// TIA Portal V20 export
DATA_BLOCK "ProdDataSimulation"   // DB5
{ DB_Accessible_From_OPC_UA := 'FALSE' }
// stored: DBAccessibleFromOPCUA false, DBAccessibleFromWebserver false, MemoryReserve 100
   VAR
      ProdDataCounter { ExternalAccessible := 'False'; ExternalVisible := 'False'; ExternalWritable := 'False'} : Struct   // Test tag prod data
         ProdDataCounter1Up1 : Bool;   // Test tag prod data
         ProdDataCounter1Up2 : Bool;   // Test tag prod data
         ProdDataCounter1Down1 : Bool;   // Test tag prod data
         ProdDataCounter1Down2 : Bool;   // Test tag prod data
         ProdDataCounter1Reset1 : Bool;   // Test tag prod data
         ProdDataCounter1Reset2 : Bool;   // Test tag prod data
         ProdDataCounter1ResetAll : Bool;   // Test tag prod data
         ProdDataCounter2Up1 : Bool;
         ProdDataCounter2Up2 : Bool;
         ProdDataCounter2Down1 : Bool;
         ProdDataCounter2Down2 : Bool;
         ProdDataCounter2Reset1 : Bool;
         ProdDataCounter2Reset2 : Bool;
         ProdDataCounter2ResetAll : Bool;
         userInterfaceVisibilityDataSet2Counter : DWord := 2#0000_0000_0000_0000_0000_0000_0000_0011;
         userInterfaceVisibilityDataSet1Counter : DWord := 2#0000_0000_0000_0000_0011_1111_1111_1111;
         ProdDataEnable : Bool;
      END_STRUCT;
      ProdDataCyclic { ExternalAccessible := 'False'; ExternalVisible := 'False'; ExternalWritable := 'False'} : Struct   // Test tag prod data
         cycleTimer1Run1 : Bool;   // Test tag prod data
         cycleTimer1Run2 : Bool;   // Test tag prod data
         cycleTimer1Hold1 : Bool;   // Test tag prod data
         cycleTimer1Hold2 : Bool;   // Test tag prod data
         cycleTimer1Reset1 : Bool;   // Test tag prod data
         cycleTimer1Reset2 : Bool;   // Test tag prod data
         cycleTimer1ResetAll : Bool;   // Test tag prod data
         cycleTimer2Run1 : Bool;   // Test tag prod data
         cycleTimer2Run2 : Bool;   // Test tag prod data
         cycleTimer2Hold1 : Bool;   // Test tag prod data
         cycleTimer2Hold2 : Bool;   // Test tag prod data
         cycleTimer2Reset1 : Bool;   // Test tag prod data
         cycleTimer2Reset2 : Bool;   // Test tag prod data
         cycleTimer2ResetAll : Bool;   // Test tag prod data
         cyclicTimerEnable : Bool;
         userInterfaceVisibilityDataSet1Cyclic : DWord := 2#0000_0000_0000_0000_0000_0000_0000_0111;
         userInterfaceVisibilityDataSet2Cyclic : DWord := 2#0000_0000_0000_0000_0000_0000_0000_0111;
         userInterfaceVisibilityDataSet3Cyclic : DWord := 2#0000_0000_0000_0000_0000_0000_1110_1111;
         userInterfaceVisibilityDataSet4Cyclic : DWord := 2#0000_0000_0000_0000_0011_1110_1111_1011;
         userInterfaceVisibilityDataSet5Cyclic : DWord := 2#0000_0000_0000_1111_1110_1111_1111_0111;
         userInterfaceVisibilityDataSet6Cyclic : DWord := 2#0000_0000_0000_0111_1111_1101_1111_1111;
         userInterfaceVisibilityDataSet7Cyclic : DWord := 2#0000_0000_0000_0000_0000_0000_0000_1111;
         userInterfaceVisibilityDataSet8Cyclic : DWord := 2#0000_0000_0000_0000_0000_0000_0000_1111;
         userInterfaceVisibilityDataSet9Cyclic : DWord := 2#0000_0000_0000_0000_0000_0000_0000_1111;
         userInterfaceVisibilityDataSet10Cyclic : DWord := 2#0000_0000_0000_0000_0000_0000_0000_1111;
         userInterfaceVisibilityDataSet11Cyclic : DWord := 2#0000_0000_0000_0000_0000_0000_0000_1111;
         userInterfaceVisibilityDataSet12Cyclic : DWord := 2#0000_0000_0000_0000_0000_0000_0000_1111;
         userInterfaceVisibilityDataSet13Cyclic : DWord := 2#0000_0000_0000_0000_0000_0000_0000_0111;
         userInterfaceVisibilityDataSet14Cyclic : DWord := 2#0000_0000_0000_0000_0000_0000_0000_1111;
      END_STRUCT;
      ProdDataLimitValues { ExternalAccessible := 'False'; ExternalVisible := 'False'; ExternalWritable := 'False'} : Struct   // Test tag prod data
         limitVal1Count1PreWarn1 : Bool;   // Test tag prod data
         limitVal1Count1PreWarn3 : Bool;   // Test tag prod data
         limitVal1Count1PreWarn2 : Bool;   // Test tag prod data
         limitVal1Count1Alarm1 : Bool;   // Test tag prod data
         limitVal1Count1Alarm3 : Bool;   // Test tag prod data
         limitVal1Count1Alarm2 : Bool;   // Test tag prod data
         limitVal1Count1 : Bool;   // Test tag prod data
         limitVal1Count2 : Bool;   // Test tag prod data
         limitVal1Count3 : Bool;   // Test tag prod data
         limitVal1Set1 : Bool;   // Test tag prod data
         limitVal1Set3 : Bool;   // Test tag prod data
         limitVal1Set2 : Bool;   // Test tag prod data
         limitValuesEnable : Bool;
         userInterfaceVisibilityDataSet2LimitValues : DWord := 2#0000_0000_0000_0000_0000_0011_1111_1111;
         userInterfaceVisibilityDataSet1LimitValues : DWord := 2#0000_0000_0000_0000_0000_0000_0000_1111;
      END_STRUCT;
      ProdDataShiftCounter { ExternalAccessible := 'False'; ExternalVisible := 'False'; ExternalWritable := 'False'} : Struct   // Test tag prod data
         shiftCounter1Cnt1Curr : Bool;   // Test tag prod data
         shiftCounter1Cnt1CurrOk : Bool;   // Test tag prod data
         shiftCounter1Cnt2Curr : Bool;   // Test tag prod data
         shiftCounter1Cnt2CurrOk : Bool;   // Test tag prod data
         shiftCounter1Cnt3Curr : Bool;   // Test tag prod data
         shiftCounter1Cnt3CurrOk : Bool;   // Test tag prod data
         shiftCounter1ResetAllExt : Bool;   // Test tag prod data
         ShiftCounterEnable : Bool;
         userInterfaceVisibilityDataSet2ShiftCounter : DWord := 2#0000_0000_0000_0000_0000_0011_1111_1111;
         userInterfaceVisibilityDataSet1ShiftCounter : DWord := 2#0000_0000_0000_0000_0000_0000_0000_1111;
      END_STRUCT;
      ProdDataShiftCounterOEE { ExternalAccessible := 'False'; ExternalVisible := 'False'; ExternalWritable := 'False'} : Struct   // Test tag prod data
         ShiftCounterOEEEnable : Bool;
         userInterfaceVisibilityDataSet2ShiftCounterOEE : DWord := 2#0000_0000_0000_0000_0000_0011_1111_1111;
         userInterfaceVisibilityDataSet1ShiftCounterOEE : DWord := 2#0000_0000_0000_0000_0000_0000_0000_1111;
      END_STRUCT;
   END_VAR
BEGIN
END_DATA_BLOCK
